FUNCTION_BLOCK DoorSensors
VAR_INPUT
END_VAR
VAR_OUTPUT
END_VAR
VAR
	r_doorCloseTimer : TON;
	r_doorOpenError : BOOL;
END_VAR

r_doorOpenError := FALSE;

IF NOT GVL_1.i_bDoorClosed THEN
    r_doorCloseTimer(IN := TRUE, PT := T#5S);
    
    IF r_doorCloseTimer.Q THEN
        r_doorOpenError := TRUE;
		r_doorCloseTimer(IN := FALSE);
    END_IF
ELSE
    r_doorCloseTimer(IN := FALSE);
    r_doorOpenError := FALSE;
END_IF
IF r_doorOpenError THEN
    GVL_1.q_bMoveUp := FALSE;
    GVL_1.q_bMoveDown := FALSE;
END_IF

END_FUNCTION_BLOCK

(* stored: Version 1.1.0.1, ProductVersion 3.1.4024.15
   POU DoorSensors: Id {9e4808e7-8ea8-415f-8fd8-6a43c03afe6b}, SpecialFunc None *)
